ABB RobotStudio station: Ajuste Cajas.rsstn

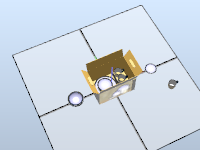
Station Station (saved by RobotStudio 20.4.9280.0)
Layout (positions relative to the parent item):
  - PlatoPando [part] at (-87.17, -4.59, 13.06) mm, rotated rx 89.99 ry -0.59 rz 2.17 deg
  - Box [graphiccomponentgroup] at (-3.94, -4.43, 4.2) mm, rotated rx 0.01 ry -0.59 rz -0.13 deg
    - PackageBox [part] at (0, 0, 0) mm, rotated rx 90 ry 0 rz 180 deg
    - Pieza_1 [part] at (89.67, -0.12, 0) mm
  - Platillo [part] at (587.41, -1.22, 1.25) mm, rotated rx 90 ry 0 rz -1.37 deg
  - PlatoHondo [part] at (-499.68, 0.5, 4.09) mm, rotated rx 90 ry 0 rz -0.39 deg
  - PlatoPando_2 [part] at (-81.29, 0.56, 24.66) mm, rotated rx 90.38 ry -0.85 rz 0.72 deg
  - PlatoPostre [part] at (-87.73, -4.54, 60.43) mm, rotated rx 89.5 ry 0.11 rz -1.62 deg
  - Pocillo [part] at (151.86, -99.78, 4.97) mm, rotated rx 90.27 ry -1.16 rz 2.85 deg
  - PlatoPando_3 [part] at (-78.57, -0.73, 36.17) mm, rotated rx 90.29 ry -0.89 rz 0.55 deg
  - PlatoPando_4 [part] at (-79.69, -1.45, 47.62) mm, rotated rx 90.24 ry -0.66 rz 0.41 deg
  - PlatoHondo_2 [part] at (-498.82, -0.6, 38.78) mm, rotated rx 89.54 ry -0.4 rz 0.27 deg
  - PlatoPostre_2 [part] at (-92.67, -11.1, 72.19) mm, rotated rx 87.36 ry 1.39 rz -4.62 deg
  - PlatoPostre_3 [part] at (-92.11, -9.86, 83.92) mm, rotated rx 87.58 ry 1.4 rz -3.9 deg
  - PlatoPostre_4 [part] at (-89.81, 0.55, 95.25) mm, rotated rx 90.62 ry 1.03 rz -0.48 deg
  - Pocillo_2 [part] at (152.85, 107.49, 4.96) mm, rotated rx 90.24 ry -0.89 rz 1.06 deg
  - Pocillo_3 [part] at (152.1, 1.81, 5.01) mm, rotated rx 89.93 ry -0.99 rz 1.46 deg
  - Pocillo_4 [part] at (698.67, -345.67, 4.12) mm, rotated rx 90 ry 0 rz -0.21 deg
